ABB RobotStudio station: Instrucciones_FOR_WHILE.rsstn

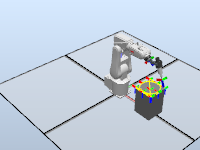
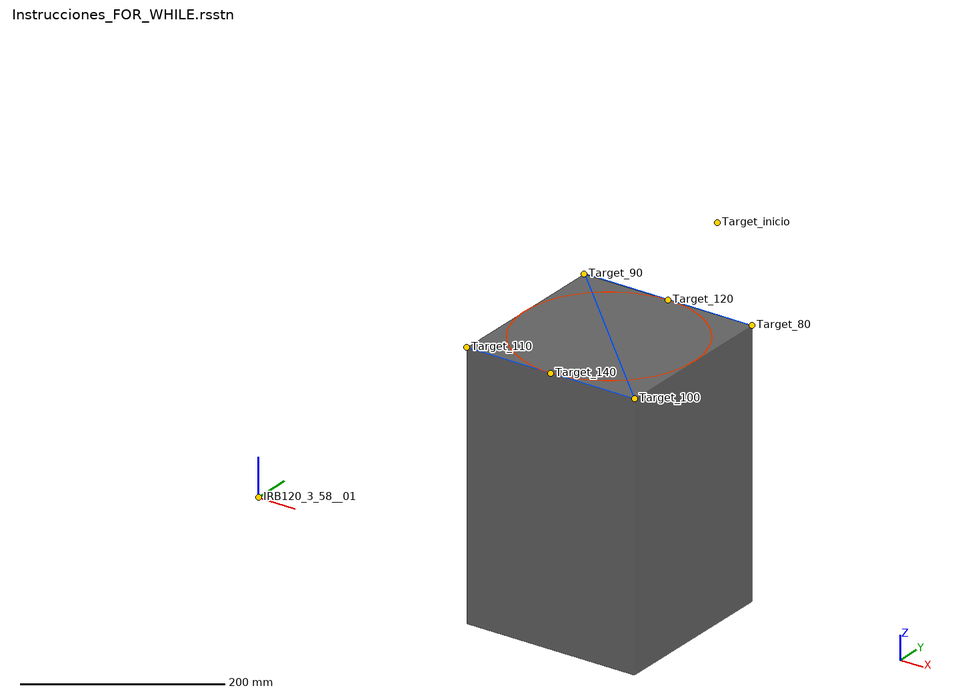
[picture v1: parts stored in the station drawn from their meshes, with robot base, taught points and paths (robot models come from the ABB library and are not in the file)]
Station P23 (saved by RobotStudio 21.2.9526.0)
Controller Controlador2
  mechanical unit ROB_1: IRB120_3_58__01, 6 joints, base frame (0, 0, 0) mm
Layout (positions relative to the parent item):
  - IRB120_3_58__01 [mechanism, from Robots\IRB120_3_58_G_01.rslib] at (0, 0, 0) mm; joint values [0, 0, 0, 0, 0.5236, 0] (rad or m)
  - MyTool [mechanism, from Training Objects\myTool.rslib] at (364.35, 0, 594) mm, rotated rx 180 ry 60 rz 180 deg
  - Pieza_2 [part] at (327.83, -113.44, 0) mm, size 200 x 200 x 300 mm
Attachment: MyTool is attached to IRB120_3_58__01 / Link6
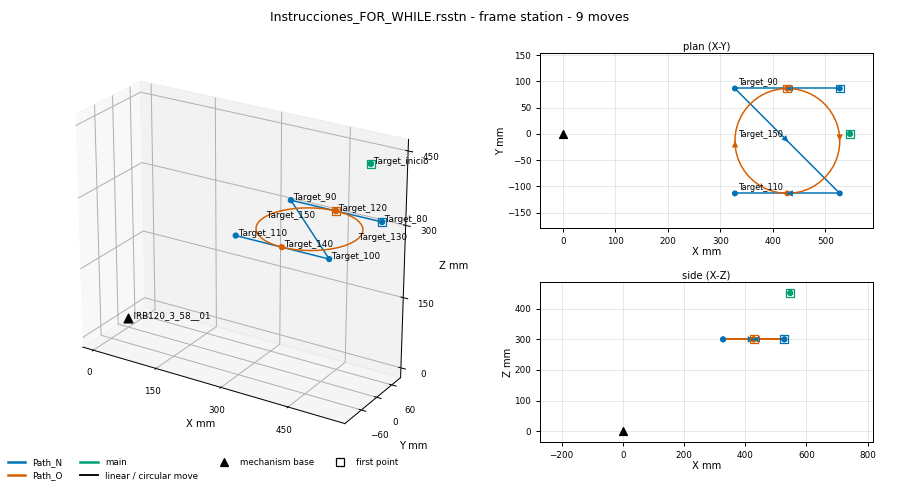
[picture p0: tool path of Instrucciones_FOR_WHILE.rsstn in frame station, 9 of 9 moves have a stored position in this frame; points joined in program order, loops and branches not executed]
Targets, tools, work objects and paths stored in the station, written as RAPID:
! task T_ROB1
MODULE CalibData
  PERS tooldata MyTool:=[TRUE,[[31.792631019,0,229.638935148],[0.945518576,0,0.325568154,0]],[1,[0,0,1],[1,0,0,0],0,0,0]];
  TASK PERS wobjdata CAJA:=[FALSE,TRUE,"",[[0,0,0],[1,0,0,0]],[[0,0,0],[1,0,0,0]]];
ENDMODULE

! task T_ROB1
MODULE Module1
  CONST robtarget Target_80:=[[527.83,86.564,300],[0,0,1,0],[0,0,0,0],[9E+09,9E+09,9E+09,9E+09,9E+09,9E+09]];
  CONST robtarget Target_90:=[[327.83,86.564,300],[0,0,1,0],[0,-1,0,0],[9E+09,9E+09,9E+09,9E+09,9E+09,9E+09]];
  CONST robtarget Target_100:=[[527.83,-113.436,300],[0,0,1,0],[-1,0,-1,0],[9E+09,9E+09,9E+09,9E+09,9E+09,9E+09]];
  CONST robtarget Target_110:=[[327.83,-113.436,300],[0,0,1,0],[-1,0,-1,0],[9E+09,9E+09,9E+09,9E+09,9E+09,9E+09]];
  CONST robtarget Target_120:=[[427.83,86.564,300],[0,0,1,0],[0,0,0,0],[9E+09,9E+09,9E+09,9E+09,9E+09,9E+09]];
  CONST robtarget Target_130:=[[527.83,-13.436,300],[0,0,1,0],[-1,0,-1,0],[9E+09,9E+09,9E+09,9E+09,9E+09,9E+09]];
  CONST robtarget Target_140:=[[427.83,-113.436,300],[0,0,1,0],[-1,0,-1,0],[9E+09,9E+09,9E+09,9E+09,9E+09,9E+09]];
  CONST robtarget Target_150:=[[327.83,-13.436,300],[0,0,1,0],[-1,0,-1,0],[9E+09,9E+09,9E+09,9E+09,9E+09,9E+09]];
  CONST robtarget Target_160:=[[452.839027956,-41.183002809,300.925979415],[0,0,1,0],[-1,0,-1,0],[9E+09,9E+09,9E+09,9E+09,9E+09,9E+09]];
  CONST robtarget Target_inicio:=[[547.330665099,0,451.64730631],[0.190808996,0,0.981627183,0],[0,0,0,0],[9E+09,9E+09,9E+09,9E+09,9E+09,9E+09]];
  PROC Path_N()
    MoveL Target_80,v1000,fine,MyTool\WObj:=CAJA;
    MoveL Target_90,v1000,fine,MyTool\WObj:=CAJA;
    MoveL Target_100,v1000,fine,MyTool\WObj:=CAJA;
    MoveL Target_110,v1000,fine,MyTool\WObj:=CAJA;
  ENDPROC
  PROC Path_O()
    MoveL Target_120,v1000,fine,MyTool\WObj:=CAJA;
    MoveC Target_130,Target_140,v1000,fine,MyTool\WObj:=CAJA;
    MoveC Target_150,Target_120,v1000,fine,MyTool\WObj:=CAJA;
  ENDPROC
  PROC main()
    MoveL Target_inicio,v1000,z100,MyTool\WObj:=wobj0;
    Path_N;
    Path_O;
    WaitTime 1;
    MoveL Target_inicio,v1000,z100,MyTool\WObj:=wobj0;
  ENDPROC
ENDMODULE

